PROGRAM MAIN
VAR
	
	RUNNING : BOOL := TRUE;
	STOPPING : BOOL := FALSE;
	
END_VAR

END_PROGRAM

(* stored: Version 1.1.0.1, ProductVersion 3.1.0.36
   POU MAIN: Id {1feaa944-c5d9-44e8-97bf-2597a802f434}, SpecialFunc None *)
